PROGRAM MAIN
VAR
	PWM1: PWM;
	tTime2: LTIME;
	a1: LREAL;
END_VAR

aoutput1:=32767;
a1:=FUN_ITR(N:=ainput1 );
tTime2:=LREAL_TO_LTIME(a1);
PWM1(bVar:=binput1 , tTime:=tTime2, Led1=>boutput1 );
pwm1.Led1;

END_PROGRAM

(* stored: Version 1.1.0.1, ProductVersion 3.1.4022.16
   POU MAIN: Id {1157e777-fbfa-498c-980e-2b883f4e682e}, SpecialFunc None *)
